Staubli VAL3: find.pgx

public program find(string& x_sItem[], bool& x_bFound[])
begin
  // check if the item has been found
  x_bFound=isDefined(pt:tTraj[x_sItem])
end
